FUNCTION_BLOCK F_LIMIT (* limiter *)
  PACKAGE iec61131::selection;
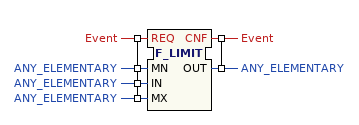
  EVENT_INPUT
    REQ WITH MN, MX, IN; (* Service Request *)
  END_EVENT
  EVENT_OUTPUT
    CNF WITH OUT; (* Confirmation of Requested Service *)
  END_EVENT
  VAR_INPUT
    MN : ANY_ELEMENTARY; (* Minimum *)
    IN : ANY_ELEMENTARY; (* Input *)
    MX : ANY_ELEMENTARY; (* Maximum *)
  END_VAR
  VAR_OUTPUT
    OUT : ANY_ELEMENTARY; (* Limited input *)
  END_VAR
END_FUNCTION_BLOCK
